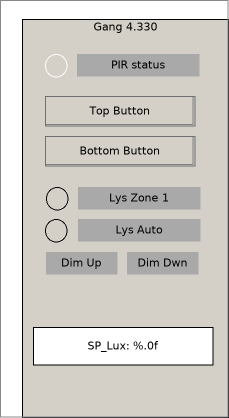
VISUALIZATION Visualization_4_330_1_1_2_1  // 229x418
    RoundedRectangle (22,19 207x399), "Gang 4.330"
    Rectangle (33,327 180x38), "SP_Lux: %.0f", text variable: P_Gang_2_143A.arrfbLysGruppe[1].fbLightCtrl.fLuxZone1
    Button (45,96 150x30), "Top Button"
        tap P_Gang_2_143A.bTopButtonZone1_Visu
    Button (45,136 150x30), "Bottom Button"
        tap P_Gang_2_143A.bBottomButtonZone1_Visu
    Ellipse (46,187 22x23), colour toggle: P_Gang_2_143A.fbLys.fbLightCtrl.bOnZone1
    Rectangle (78,187 122x22), "Lys Zone 1"
    Rectangle (46,252 71x22), "Dim Up", colour toggle: P_Gang_2_143A.arrfbLysGruppe[1].fbLightCtrl.bDimUp
    Rectangle (127,252 71x22), "Dim Dwn", colour toggle: P_Gang_2_143A.arrfbLysGruppe[1].fbLightCtrl.bDimDwn
    Ellipse (45,219 22x23), colour toggle: P_Gang_2_143A.arrfbLysGruppe[1].fbLightCtrl.bAutoZone1
    Rectangle (78,219 122x22), "Lys Auto"
    Ellipse (45,54 22x23), colour toggle: P_Gang_2_143A.arrfbLysGruppe[1].fbLightCtrl.bPIR
    Rectangle (77,54 122x22), "PIR status"
END_VISUALIZATION

(* stored: Version 1.1.0.1
   Visu Visualization_4_330_1_1_2_1: Id {00e4842d-f611-48e6-838e-5f218c5d8238} *)
